FUNCTION_BLOCK ExtensionBase EXTENDS Disposable IMPLEMENTS I_Extension
VAR
	_name : T_MAXSTRING;
	eventEmitter : EventEmitter;
	inputPortHost : InputPortHost(eventEmitter);
	outputPortHost : OutputPortHost(eventEmitter);
	parameterHost : ParameterHost(eventEmitter);
	contentHost : ContentHost(eventEmitter);
	errorHost : ErrorHost(eventEmitter);
	metadataHost : MetadataHost(eventEmitter);
END_VAR

METHOD PUBLIC Accept
VAR_INPUT
	Visitor : I_ExtensionVisitor;
END_VAR
Visitor.VisitExtension(this^);
END_METHOD

METHOD AddContent
VAR_INPUT
	Content : I_Content;
END_VAR
contentHost.AddContent(Content);
END_METHOD

METHOD PUBLIC AddDataAsContent : I_Content;
VAR_INPUT
	Name : T_MAXSTRING;
	Data : I_Datatype;
END_VAR
AddDataAsContent := contentHost.AddDataAsContent(Name, Data);
END_METHOD

METHOD PUBLIC AddDataAsInputPort : I_InputPort;
VAR_INPUT
	Name : T_MAXSTRING;
	Data : I_Datatype;
END_VAR
AddDataAsInputPort := inputPortrHost.AddDataAsInputPort(Name, Data);
END_METHOD

METHOD PUBLIC AddDataAsMetadata : I_Metadata;
VAR_INPUT
	Name : T_MAXSTRING;
	Data : I_Datatype;
END_VAR
AddDataAsMetadata := metadataHost.AddDataAsMetadata(Name, Data);
END_METHOD

METHOD PUBLIC AddDataAsOutputPort : I_OutputPort;
VAR_INPUT
	Name : T_MAXSTRING;
	Data : I_Datatype;
END_VAR
AddDataAsOutputPort := outputPortrHost.AddDataAsOutputPort(Name, Data);
END_METHOD

METHOD PUBLIC AddDataAsParameter : I_Parameter;
VAR_INPUT
	Name : T_MAXSTRING;
	Data : I_Datatype;
END_VAR
AddDataAsParameter := parameterHost.AddDataAsParameter(Name, Data);
END_METHOD

METHOD AddError
VAR_INPUT
	Error : I_Error;
END_VAR
errorHost.AddError(Error);
END_METHOD

METHOD AddInputPort
VAR_INPUT
	InputPort : I_InputPort;
END_VAR
inputPortHost.AddInputPort(InputPort);
END_METHOD

METHOD AddMetadata
VAR_INPUT
	Metadata : I_Metadata;
END_VAR
metadataHost.AddMetadata(Metadata);
END_METHOD

METHOD AddOutputPort
VAR_INPUT
	OutputPort : I_OutputPort;
END_VAR
outputPortHost.AddOutputPort(OutputPort);
END_METHOD

METHOD AddParameter
VAR_INPUT
	Parameter : I_Parameter;
END_VAR
parameterHost.AddParameter(Parameter);
END_METHOD

METHOD FB_init : BOOL
VAR_INPUT
	bInitRetains : BOOL; // if TRUE, the retain variables are initialized (warm start / cold start)
	bInCopyCode : BOOL;  // if TRUE, the instance afterwards gets moved into the copy code (online change)
	Name : T_MAXSTRING;
END_VAR
_name := Name;
InitializeExtension(THIS^);
END_METHOD

METHOD PROTECTED InitializeExtension
VAR_INPUT
	Self : I_Extension;
END_VAR
END_METHOD

PROPERTY PUBLIC Name : T_MAXSTRING
GET
Name := _name;
END_GET
END_PROPERTY

METHOD PUBLIC OffEvent
VAR_INPUT
	EventName : T_MaxString;
	EventHandler : I_EventHandler;
END_VAR
eventEmitter.OffEvent(EventName, EventHandler);
END_METHOD

METHOD PUBLIC OnceEvent
VAR_INPUT
	EventName : T_MaxString;
	EventHandler : I_EventHandler;
END_VAR
eventEmitter.OnceEvent(EventName, EventHandler);
END_METHOD

METHOD PUBLIC OnEvent
VAR_INPUT
	EventName : T_MaxString;
	EventHandler : I_EventHandler;
END_VAR
eventEmitter.OnEvent(EventName, EventHandler);
END_METHOD

METHOD PUBLIC SerializeWith
VAR_INPUT
	Serializer : I_Serializer;
END_VAR
Serializer.StartObject();
inputPortHost.SerializeWith(Serializer);
outputPortHost.SerializeWith(Serializer);
parameterHost.SerializeWith(Serializer);
contentHost.SerializeWith(Serializer);
errorHost.SerializeWith(Serializer);
metadataHost.SerializeWith(Serializer);
Serializer.EndObject();
END_METHOD

METHOD PUBLIC TryDeserializeFrom : BOOL
VAR_INPUT
	Deserializer : I_Deserializer;
END_VAR
TryDeserializeFrom := parameterHost.TryDeserializeFrom(Deserializer);
END_METHOD

METHOD PUBLIC TryGetContentByName : BOOL
VAR_INPUT
	Name : T_MAXSTRING;
	Destination : REFERENCE TO I_Content;
END_VAR
TryGetContentByName := contentHost.TryGetContentByName(Name,Destination);
END_METHOD

METHOD PUBLIC TryGetInputPortByName : BOOL
VAR_INPUT
	Name : T_MAXSTRING;
	Destination : REFERENCE TO I_InputPort;
END_VAR
TryGetInputPortByName := inputPortHost.TryGetInputPortByName(Name,Destination);
END_METHOD

METHOD PUBLIC TryGetMetadataByName : BOOL
VAR_INPUT
	Name : T_MAXSTRING;
	Destination : REFERENCE TO I_Metadata;
END_VAR
TryGetMetadataByName := metadataHost.TryGetMetadataByName(Name,Destination);
END_METHOD

METHOD PUBLIC TryGetOutputPortByName : BOOL
VAR_INPUT
	Name : T_MAXSTRING;
	Destination : REFERENCE TO I_OutputPort;
END_VAR
TryGetOutputPortByName := outputPortHost.TryGetOutputPortByName(Name,Destination);
END_METHOD

METHOD PUBLIC TryGetParameterByName : BOOL
VAR_INPUT
	Name : T_MAXSTRING;
	Destination : REFERENCE TO I_Parameter;
END_VAR
TryGetParameterByName := parameterHost.TryGetParameterByName(Name,Destination);
END_METHOD

END_FUNCTION_BLOCK

(* stored: Version 1.1.0.1, ProductVersion 3.1.4024.12
   POU ExtensionBase: Id {42104a2a-bb11-0099-07c8-1566fddf2573}, SpecialFunc None
   Folder Constructor: Id {fef26075-0f2d-0849-2106-d8875bfcef87}
   Folder Protected: Id {8929ae02-54e4-48f4-9cde-455bb332213a}
   Method Accept: Id {c7a8469c-4655-04f0-2d46-e58992b2a552}
   Method AddContent: Id {6ea2b1d8-d6b2-4d47-b550-47d68cad2d2c}
   Method AddDataAsContent: Id {e881ed24-909b-4499-854b-919db48b9f56}
   Method AddDataAsInputPort: Id {a0b99e5f-97a0-4cb4-85b1-be3501128a16}
   Method AddDataAsMetadata: Id {d53f29f1-b79b-4bd5-bcc5-e393812fb6bd}
   Method AddDataAsOutputPort: Id {0a62794b-674a-488d-bb99-70710b5485e8}
   Method AddDataAsParameter: Id {208dca8c-4c22-45b1-a6b5-b665342594b4}
   Method AddError: Id {25dc5072-bec6-4adc-b2cf-46ff0174bb16}
   Method AddInputPort: Id {9e63d406-abf0-4693-b057-e8bdf718d997}
   Method AddMetadata: Id {47801752-9488-4924-95cc-3210bc37bfa4}
   Method AddOutputPort: Id {53427e17-c470-45c4-8203-d9e21c021e85}
   Method AddParameter: Id {23dd46d8-4d23-4b8e-a814-7bae28ecf1e9}
   Method FB_init: Id {b8dc459b-fb89-0be1-1d4e-1dd2490364b6}
   Method InitializeExtension: Id {c523b599-657c-48d8-9a15-a024d5cd3cac}
   Property Name: Id {3ea0ca14-7e1c-0f9c-0dd4-fc640a163eef}
   Get Get: Id {89da2b88-6436-0494-1a12-900ee5d5f448}
   Method OffEvent: Id {7c991add-898b-4ce2-b48c-156ceb4e3445}
   Method OnceEvent: Id {057d5c02-4afe-46f3-b0ee-2a2800b6229d}
   Method OnEvent: Id {84177a9d-8640-40f8-aff3-a509bb613f25}
   Method SerializeWith: Id {f0a208e7-7dd4-4f99-8c68-aad6715feaed}
   Method TryDeserializeFrom: Id {6d59da26-ba4e-4a2b-89b3-fd3987fd40bc}
   Method TryGetContentByName: Id {6ca9fed6-43c8-42ca-90d1-dc23b9a9178a}
   Method TryGetInputPortByName: Id {989b9f1f-f3dc-4265-a126-3564404c6f91}
   Method TryGetMetadataByName: Id {79a0c769-c359-4c92-9cee-f8085d22fa56}
   Method TryGetOutputPortByName: Id {d210715a-df61-446a-bbe4-68c40d5deede}
   Method TryGetParameterByName: Id {df6993d6-fa50-494d-8b42-4f0d28a492f0} *)
